{attribute 'strict'}
TYPE E_RecipesManagerStateCreateRemove :
(
	RECIPES_MANAGER_CREATE_REMOVE_OPERATION 			:= 0,	(* Create/Remove recipe with selected name *)
	RECIPES_MANAGER_CREATE_REMOVE_GET_RECIPES_COUNT 	:= 10,	(* Getting number of detected recipes in directory *)
	RECIPES_MANAGER_CREATE_REMOVE_RELOAD				:= 20,	(* Reloading recipes manager *)
	RECIPES_MANAGER_CREATE_REMOVE_GET_RECIPES_NAMES 	:= 30,	(* Getting names of recipes in selected directory *)
	RECIPES_MANAGER_CREATE_REMOVE_GET_VARIABLE_NAMES	:= 40,	(* Getting names of variables from recipes manager *)
	RECIPES_MANAGER_CREATE_REMOVE_GET_VARIABLE_VALUES	:= 50,	(* Getting variable values from selected recipe *)
	RECIPES_MANAGER_CREATE_REMOVE_DONE					:= 60	(* Removing selected recipe *)
);
END_TYPE

(* stored: Version 1.1.0.1, ProductVersion 3.1.4024.12
   DUT E_RecipesManagerStateCreateRemove: Id {4b5e00b2-39fe-46c5-9cf3-b722ce066860} *)
